Fanuc TP program (LS listing): MOVE2LOAD.LS

/PROG  MOVE2LOAD
/ATTR
OWNER		= MNEDITOR;
COMMENT		= "macro load pt";
PROG_SIZE	= 279;
CREATE		= DATE 19-09-30  TIME 15:32:40;
MODIFIED	= DATE 19-09-30  TIME 15:42:48;
FILE_NAME	= PROGRAM_;
VERSION		= 0;
LINE_COUNT	= 4;
MEMORY_SIZE	= 635;
PROTECT		= READ_WRITE;
TCD:  STACK_SIZE	= 0,
      TASK_PRIORITY	= 50,
      TIME_SLICE	= 0,
      BUSY_LAMP_OFF	= 0,
      ABORT_REQUEST	= 0,
      PAUSE_REQUEST	= 0;
DEFAULT_GROUP	= 1,*,*,*,*;
CONTROL_CODE	= 00000000 00000000;
/APPL
/APPL

AUTO_SINGULARITY_HEADER;
  ENABLE_SINGULARITY_AVOIDANCE   : TRUE;
/MN
   1:  !Set UT & UF ;
   2:  UTOOL_NUM=1 ;
   3:  UFRAME_NUM=2 ;
   4:L PR[2:LOAD PT] 250mm/sec FINE    ;
/POS
/END
